{attribute 'Tc2GvlVarNames'}
VAR_GLOBAL
	eCodeAIType							: E_CodeAIType;
	


END_VAR

(* stored: Version 1.1.0.1
   GVL CodeAI: Id {0be59666-1934-4ac9-a7db-3bbdec11e330} *)
